// TIA Portal V16 export
// export: Created 2023-03-29T11:03:28.4713144Z, ExportSetting WithDefaults, DisplayName Totally Integrated Automation Portal, DisplayVersion V16 Update 6, DisplayName TIA Portal Version Control Interface, DisplayVersion V16 Update 2, DisplayName TIA Portal Openness, DisplayVersion V16 Update 6, DisplayName STEP 7 Professional, DisplayVersion V16 Update 6, DisplayName STEP 7 Safety, DisplayVersion V16, DisplayName WinCC Advanced, DisplayVersion V16 Update 6
FUNCTION "Synchroniczna_wymiana_danych_PLC1-PLC2" : Void   // FC34, LAD
TITLE = Przekazywanie zmian parametrów
{ S7_Optimized_Access := 'TRUE' }
AUTHOR : rtecmer
VERSION : 0.1
// Funkcja grupuje bloki funkcji służąc wymianie danych HMI - PLC1, HMI-PLC2 i SCADA. Wprowadzanie wartości z poziomu HMI Zbiorniki lub HMI Pompownia czy SCADA jest nadpisywane w docelowym sterowniku. Zmian włónych parametrów układu sterowania pompownią, zbiornikami można dokonywać w dowolnego miejsca.
// stored: AutoNumber true, IsIECCheckEnabled false, SetENOAutomatically false, UDAEnableTagReadback false
   VAR_TEMP   // added for the SCL form of the ladder/FBD networks
      _w1 : Bool;
   END_VAR
BEGIN

REGION Network 2: Detekcja zmiany wartości nastaw - Pozim napełniania
   // Funkcja po przeprowadzeniu sprawdzenia czy nastąpiły zmiany w danych przekazuje nowe wartości
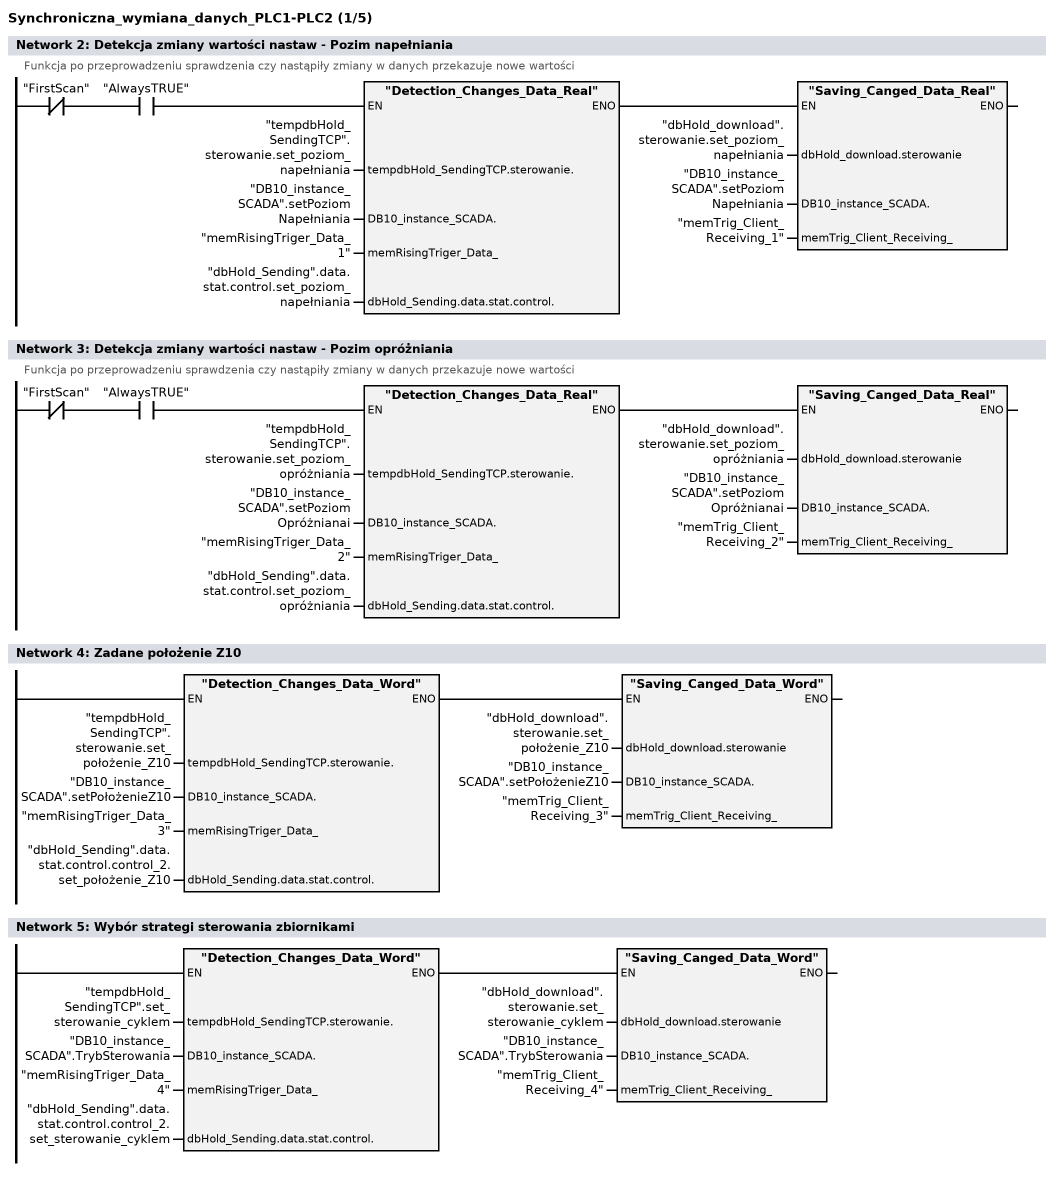
   RUNG wire#powerrail
      I_Contact( "FirstScan" )
      Contact( "AlwaysTRUE" )
      "Detection_Changes_Data_Real"("tempdbHold_SendingTCP.sterowanie." := "tempdbHold_SendingTCP".sterowanie.set_poziom_napełniania, "DB10_instance_SCADA." := "DB10_instance_SCADA".setPoziomNapełniania, memRisingTriger_Data_ := "memRisingTriger_Data_1", "dbHold_Sending.data.stat.control." := "dbHold_Sending".data.stat.control.set_poziom_napełniania)
      "Saving_Canged_Data_Real"("dbHold_download.sterowanie" := "dbHold_download".sterowanie.set_poziom_napełniania, "DB10_instance_SCADA." := "DB10_instance_SCADA".setPoziomNapełniania, memTrig_Client_Receiving_ := "memTrig_Client_Receiving_1")
   END_RUNG
   // the same network as SCL:
   "Detection_Changes_Data_Real"(EN := NOT "FirstScan" AND "AlwaysTRUE",
                           "tempdbHold_SendingTCP.sterowanie." := "tempdbHold_SendingTCP".sterowanie.set_poziom_napełniania,
                           "DB10_instance_SCADA." := "DB10_instance_SCADA".setPoziomNapełniania,
                           memRisingTriger_Data_ := "memRisingTriger_Data_1",
                           "dbHold_Sending.data.stat.control." := "dbHold_Sending".data.stat.control.set_poziom_napełniania,
                           ENO => #_w1);
   IF #_w1 THEN
       "Saving_Canged_Data_Real"("dbHold_download.sterowanie" := "dbHold_download".sterowanie.set_poziom_napełniania,
                               "DB10_instance_SCADA." := "DB10_instance_SCADA".setPoziomNapełniania,
                               memTrig_Client_Receiving_ := "memTrig_Client_Receiving_1");
   END_IF;
END_REGION

REGION Network 3: Detekcja zmiany wartości nastaw - Pozim opróżniania
   // Funkcja po przeprowadzeniu sprawdzenia czy nastąpiły zmiany w danych przekazuje nowe wartości
   RUNG wire#powerrail
      I_Contact( "FirstScan" )
      Contact( "AlwaysTRUE" )
      "Detection_Changes_Data_Real"("tempdbHold_SendingTCP.sterowanie." := "tempdbHold_SendingTCP".sterowanie.set_poziom_opróżniania, "DB10_instance_SCADA." := "DB10_instance_SCADA".setPoziomOpróżnianai, memRisingTriger_Data_ := "memRisingTriger_Data_2", "dbHold_Sending.data.stat.control." := "dbHold_Sending".data.stat.control.set_poziom_opróżniania)
      "Saving_Canged_Data_Real"("dbHold_download.sterowanie" := "dbHold_download".sterowanie.set_poziom_opróżniania, "DB10_instance_SCADA." := "DB10_instance_SCADA".setPoziomOpróżnianai, memTrig_Client_Receiving_ := "memTrig_Client_Receiving_2")
   END_RUNG
   // the same network as SCL:
   "Detection_Changes_Data_Real"(EN := NOT "FirstScan" AND "AlwaysTRUE",
                           "tempdbHold_SendingTCP.sterowanie." := "tempdbHold_SendingTCP".sterowanie.set_poziom_opróżniania,
                           "DB10_instance_SCADA." := "DB10_instance_SCADA".setPoziomOpróżnianai,
                           memRisingTriger_Data_ := "memRisingTriger_Data_2",
                           "dbHold_Sending.data.stat.control." := "dbHold_Sending".data.stat.control.set_poziom_opróżniania,
                           ENO => #_w1);
   IF #_w1 THEN
       "Saving_Canged_Data_Real"("dbHold_download.sterowanie" := "dbHold_download".sterowanie.set_poziom_opróżniania,
                               "DB10_instance_SCADA." := "DB10_instance_SCADA".setPoziomOpróżnianai,
                               memTrig_Client_Receiving_ := "memTrig_Client_Receiving_2");
   END_IF;
END_REGION

REGION Network 4: Zadane położenie Z10
   RUNG wire#powerrail
      "Detection_Changes_Data_Word"("tempdbHold_SendingTCP.sterowanie." := "tempdbHold_SendingTCP".sterowanie.set_położenie_Z10, "DB10_instance_SCADA." := "DB10_instance_SCADA".setPołożenieZ10, memRisingTriger_Data_ := "memRisingTriger_Data_3", "dbHold_Sending.data.stat.control." := "dbHold_Sending".data.stat.control.control_2.set_położenie_Z10)
      "Saving_Canged_Data_Word"("dbHold_download.sterowanie" := "dbHold_download".sterowanie.set_położenie_Z10, "DB10_instance_SCADA." := "DB10_instance_SCADA".setPołożenieZ10, memTrig_Client_Receiving_ := "memTrig_Client_Receiving_3")
   END_RUNG
   // the same network as SCL:
   "Detection_Changes_Data_Word"("tempdbHold_SendingTCP.sterowanie." := "tempdbHold_SendingTCP".sterowanie.set_położenie_Z10,
                           "DB10_instance_SCADA." := "DB10_instance_SCADA".setPołożenieZ10,
                           memRisingTriger_Data_ := "memRisingTriger_Data_3",
                           "dbHold_Sending.data.stat.control." := "dbHold_Sending".data.stat.control.control_2.set_położenie_Z10,
                           ENO => #_w1);
   IF #_w1 THEN
       "Saving_Canged_Data_Word"("dbHold_download.sterowanie" := "dbHold_download".sterowanie.set_położenie_Z10,
                               "DB10_instance_SCADA." := "DB10_instance_SCADA".setPołożenieZ10,
                               memTrig_Client_Receiving_ := "memTrig_Client_Receiving_3");
   END_IF;
END_REGION

REGION Network 5: Wybór strategi sterowania zbiornikami
   RUNG wire#powerrail
      "Detection_Changes_Data_Word"("tempdbHold_SendingTCP.sterowanie." := "tempdbHold_SendingTCP".set_sterowanie_cyklem, "DB10_instance_SCADA." := "DB10_instance_SCADA".TrybSterowania, memRisingTriger_Data_ := "memRisingTriger_Data_4", "dbHold_Sending.data.stat.control." := "dbHold_Sending".data.stat.control.control_2.set_sterowanie_cyklem)
      "Saving_Canged_Data_Word"("dbHold_download.sterowanie" := "dbHold_download".sterowanie.set_sterowanie_cyklem, "DB10_instance_SCADA." := "DB10_instance_SCADA".TrybSterowania, memTrig_Client_Receiving_ := "memTrig_Client_Receiving_4")
   END_RUNG
   // the same network as SCL:
   "Detection_Changes_Data_Word"("tempdbHold_SendingTCP.sterowanie." := "tempdbHold_SendingTCP".set_sterowanie_cyklem,
                           "DB10_instance_SCADA." := "DB10_instance_SCADA".TrybSterowania,
                           memRisingTriger_Data_ := "memRisingTriger_Data_4",
                           "dbHold_Sending.data.stat.control." := "dbHold_Sending".data.stat.control.control_2.set_sterowanie_cyklem,
                           ENO => #_w1);
   IF #_w1 THEN
       "Saving_Canged_Data_Word"("dbHold_download.sterowanie" := "dbHold_download".sterowanie.set_sterowanie_cyklem,
                               "DB10_instance_SCADA." := "DB10_instance_SCADA".TrybSterowania,
                               memTrig_Client_Receiving_ := "memTrig_Client_Receiving_4");
   END_IF;
END_REGION

REGION Network 6: Godzina start napełnianie
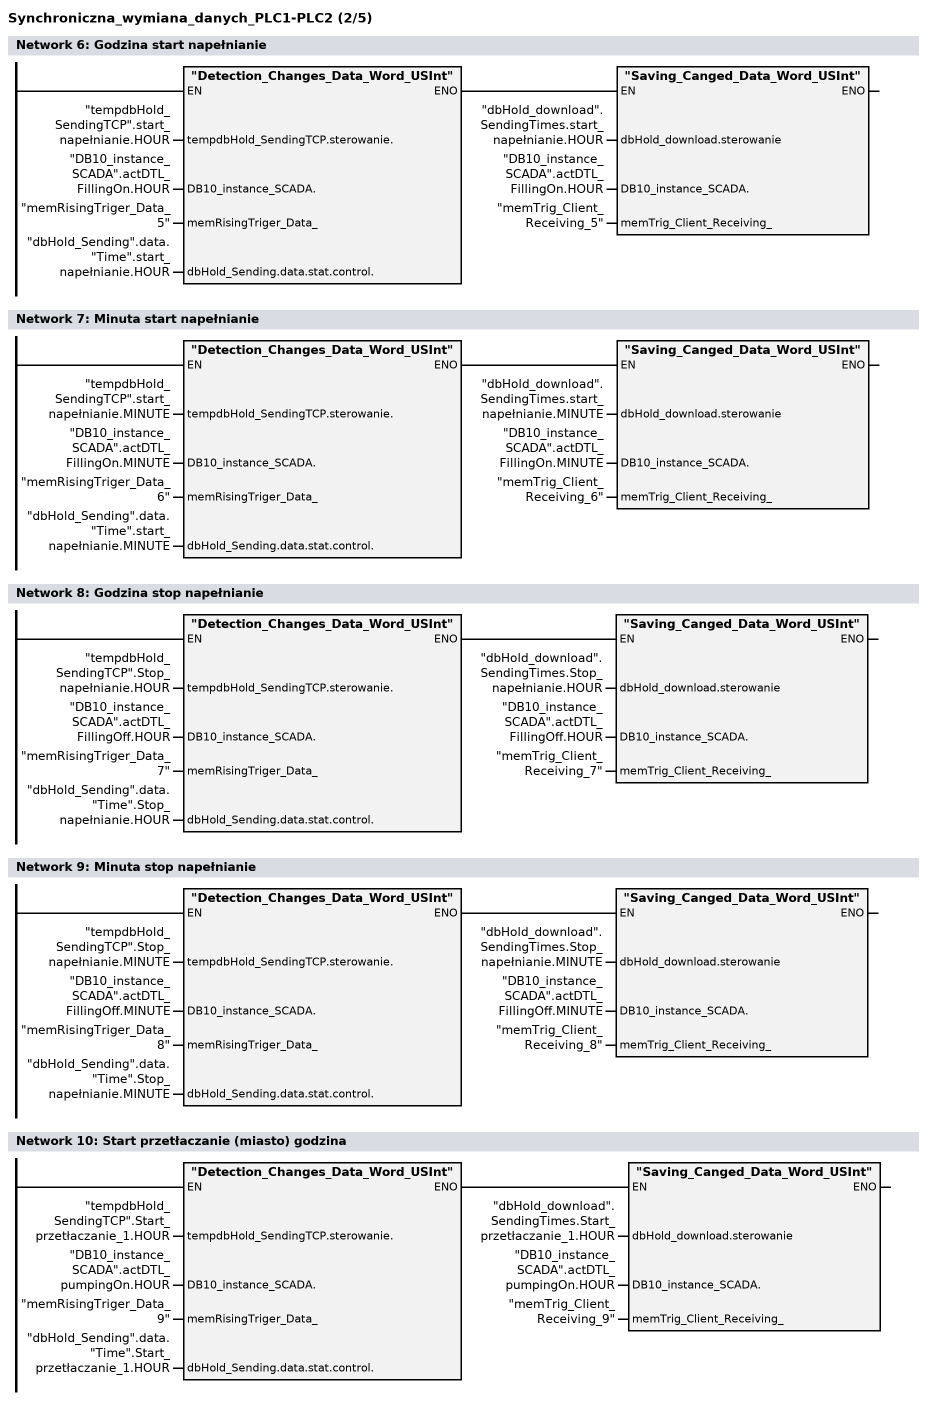
   RUNG wire#powerrail
      "Detection_Changes_Data_Word_USInt"("tempdbHold_SendingTCP.sterowanie." := "tempdbHold_SendingTCP".start_napełnianie.HOUR, "DB10_instance_SCADA." := "DB10_instance_SCADA".actDTL_FillingOn.HOUR, memRisingTriger_Data_ := "memRisingTriger_Data_5", "dbHold_Sending.data.stat.control." := "dbHold_Sending".data."Time".start_napełnianie.HOUR)
      "Saving_Canged_Data_Word_USInt"("dbHold_download.sterowanie" := "dbHold_download".SendingTimes.start_napełnianie.HOUR, "DB10_instance_SCADA." := "DB10_instance_SCADA".actDTL_FillingOn.HOUR, memTrig_Client_Receiving_ := "memTrig_Client_Receiving_5")
   END_RUNG
   // the same network as SCL:
   "Detection_Changes_Data_Word_USInt"("tempdbHold_SendingTCP.sterowanie." := "tempdbHold_SendingTCP".start_napełnianie.HOUR,
                           "DB10_instance_SCADA." := "DB10_instance_SCADA".actDTL_FillingOn.HOUR,
                           memRisingTriger_Data_ := "memRisingTriger_Data_5",
                           "dbHold_Sending.data.stat.control." := "dbHold_Sending".data."Time".start_napełnianie.HOUR,
                           ENO => #_w1);
   IF #_w1 THEN
       "Saving_Canged_Data_Word_USInt"("dbHold_download.sterowanie" := "dbHold_download".SendingTimes.start_napełnianie.HOUR,
                               "DB10_instance_SCADA." := "DB10_instance_SCADA".actDTL_FillingOn.HOUR,
                               memTrig_Client_Receiving_ := "memTrig_Client_Receiving_5");
   END_IF;
END_REGION

REGION Network 7: Minuta start napełnianie
   RUNG wire#powerrail
      "Detection_Changes_Data_Word_USInt"("tempdbHold_SendingTCP.sterowanie." := "tempdbHold_SendingTCP".start_napełnianie.MINUTE, "DB10_instance_SCADA." := "DB10_instance_SCADA".actDTL_FillingOn.MINUTE, memRisingTriger_Data_ := "memRisingTriger_Data_6", "dbHold_Sending.data.stat.control." := "dbHold_Sending".data."Time".start_napełnianie.MINUTE)
      "Saving_Canged_Data_Word_USInt"("dbHold_download.sterowanie" := "dbHold_download".SendingTimes.start_napełnianie.MINUTE, "DB10_instance_SCADA." := "DB10_instance_SCADA".actDTL_FillingOn.MINUTE, memTrig_Client_Receiving_ := "memTrig_Client_Receiving_6")
   END_RUNG
   // the same network as SCL:
   "Detection_Changes_Data_Word_USInt"("tempdbHold_SendingTCP.sterowanie." := "tempdbHold_SendingTCP".start_napełnianie.MINUTE,
                           "DB10_instance_SCADA." := "DB10_instance_SCADA".actDTL_FillingOn.MINUTE,
                           memRisingTriger_Data_ := "memRisingTriger_Data_6",
                           "dbHold_Sending.data.stat.control." := "dbHold_Sending".data."Time".start_napełnianie.MINUTE,
                           ENO => #_w1);
   IF #_w1 THEN
       "Saving_Canged_Data_Word_USInt"("dbHold_download.sterowanie" := "dbHold_download".SendingTimes.start_napełnianie.MINUTE,
                               "DB10_instance_SCADA." := "DB10_instance_SCADA".actDTL_FillingOn.MINUTE,
                               memTrig_Client_Receiving_ := "memTrig_Client_Receiving_6");
   END_IF;
END_REGION

REGION Network 8: Godzina stop napełnianie
   RUNG wire#powerrail
      "Detection_Changes_Data_Word_USInt"("tempdbHold_SendingTCP.sterowanie." := "tempdbHold_SendingTCP".Stop_napełnianie.HOUR, "DB10_instance_SCADA." := "DB10_instance_SCADA".actDTL_FillingOff.HOUR, memRisingTriger_Data_ := "memRisingTriger_Data_7", "dbHold_Sending.data.stat.control." := "dbHold_Sending".data."Time".Stop_napełnianie.HOUR)
      "Saving_Canged_Data_Word_USInt"("dbHold_download.sterowanie" := "dbHold_download".SendingTimes.Stop_napełnianie.HOUR, "DB10_instance_SCADA." := "DB10_instance_SCADA".actDTL_FillingOff.HOUR, memTrig_Client_Receiving_ := "memTrig_Client_Receiving_7")
   END_RUNG
   // the same network as SCL:
   "Detection_Changes_Data_Word_USInt"("tempdbHold_SendingTCP.sterowanie." := "tempdbHold_SendingTCP".Stop_napełnianie.HOUR,
                           "DB10_instance_SCADA." := "DB10_instance_SCADA".actDTL_FillingOff.HOUR,
                           memRisingTriger_Data_ := "memRisingTriger_Data_7",
                           "dbHold_Sending.data.stat.control." := "dbHold_Sending".data."Time".Stop_napełnianie.HOUR,
                           ENO => #_w1);
   IF #_w1 THEN
       "Saving_Canged_Data_Word_USInt"("dbHold_download.sterowanie" := "dbHold_download".SendingTimes.Stop_napełnianie.HOUR,
                               "DB10_instance_SCADA." := "DB10_instance_SCADA".actDTL_FillingOff.HOUR,
                               memTrig_Client_Receiving_ := "memTrig_Client_Receiving_7");
   END_IF;
END_REGION

REGION Network 9: Minuta stop napełnianie
   RUNG wire#powerrail
      "Detection_Changes_Data_Word_USInt"("tempdbHold_SendingTCP.sterowanie." := "tempdbHold_SendingTCP".Stop_napełnianie.MINUTE, "DB10_instance_SCADA." := "DB10_instance_SCADA".actDTL_FillingOff.MINUTE, memRisingTriger_Data_ := "memRisingTriger_Data_8", "dbHold_Sending.data.stat.control." := "dbHold_Sending".data."Time".Stop_napełnianie.MINUTE)
      "Saving_Canged_Data_Word_USInt"("dbHold_download.sterowanie" := "dbHold_download".SendingTimes.Stop_napełnianie.MINUTE, "DB10_instance_SCADA." := "DB10_instance_SCADA".actDTL_FillingOff.MINUTE, memTrig_Client_Receiving_ := "memTrig_Client_Receiving_8")
   END_RUNG
   // the same network as SCL:
   "Detection_Changes_Data_Word_USInt"("tempdbHold_SendingTCP.sterowanie." := "tempdbHold_SendingTCP".Stop_napełnianie.MINUTE,
                           "DB10_instance_SCADA." := "DB10_instance_SCADA".actDTL_FillingOff.MINUTE,
                           memRisingTriger_Data_ := "memRisingTriger_Data_8",
                           "dbHold_Sending.data.stat.control." := "dbHold_Sending".data."Time".Stop_napełnianie.MINUTE,
                           ENO => #_w1);
   IF #_w1 THEN
       "Saving_Canged_Data_Word_USInt"("dbHold_download.sterowanie" := "dbHold_download".SendingTimes.Stop_napełnianie.MINUTE,
                               "DB10_instance_SCADA." := "DB10_instance_SCADA".actDTL_FillingOff.MINUTE,
                               memTrig_Client_Receiving_ := "memTrig_Client_Receiving_8");
   END_IF;
END_REGION

REGION Network 10: Start przetłaczanie (miasto) godzina
   RUNG wire#powerrail
      "Detection_Changes_Data_Word_USInt"("tempdbHold_SendingTCP.sterowanie." := "tempdbHold_SendingTCP".Start_przetłaczanie_1.HOUR, "DB10_instance_SCADA." := "DB10_instance_SCADA".actDTL_pumpingOn.HOUR, memRisingTriger_Data_ := "memRisingTriger_Data_9", "dbHold_Sending.data.stat.control." := "dbHold_Sending".data."Time".Start_przetłaczanie_1.HOUR)
      "Saving_Canged_Data_Word_USInt"("dbHold_download.sterowanie" := "dbHold_download".SendingTimes.Start_przetłaczanie_1.HOUR, "DB10_instance_SCADA." := "DB10_instance_SCADA".actDTL_pumpingOn.HOUR, memTrig_Client_Receiving_ := "memTrig_Client_Receiving_9")
   END_RUNG
   // the same network as SCL:
   "Detection_Changes_Data_Word_USInt"("tempdbHold_SendingTCP.sterowanie." := "tempdbHold_SendingTCP".Start_przetłaczanie_1.HOUR,
                           "DB10_instance_SCADA." := "DB10_instance_SCADA".actDTL_pumpingOn.HOUR,
                           memRisingTriger_Data_ := "memRisingTriger_Data_9",
                           "dbHold_Sending.data.stat.control." := "dbHold_Sending".data."Time".Start_przetłaczanie_1.HOUR,
                           ENO => #_w1);
   IF #_w1 THEN
       "Saving_Canged_Data_Word_USInt"("dbHold_download.sterowanie" := "dbHold_download".SendingTimes.Start_przetłaczanie_1.HOUR,
                               "DB10_instance_SCADA." := "DB10_instance_SCADA".actDTL_pumpingOn.HOUR,
                               memTrig_Client_Receiving_ := "memTrig_Client_Receiving_9");
   END_IF;
END_REGION

REGION Network 11: Start przetłaczanie (miasto) mnutya
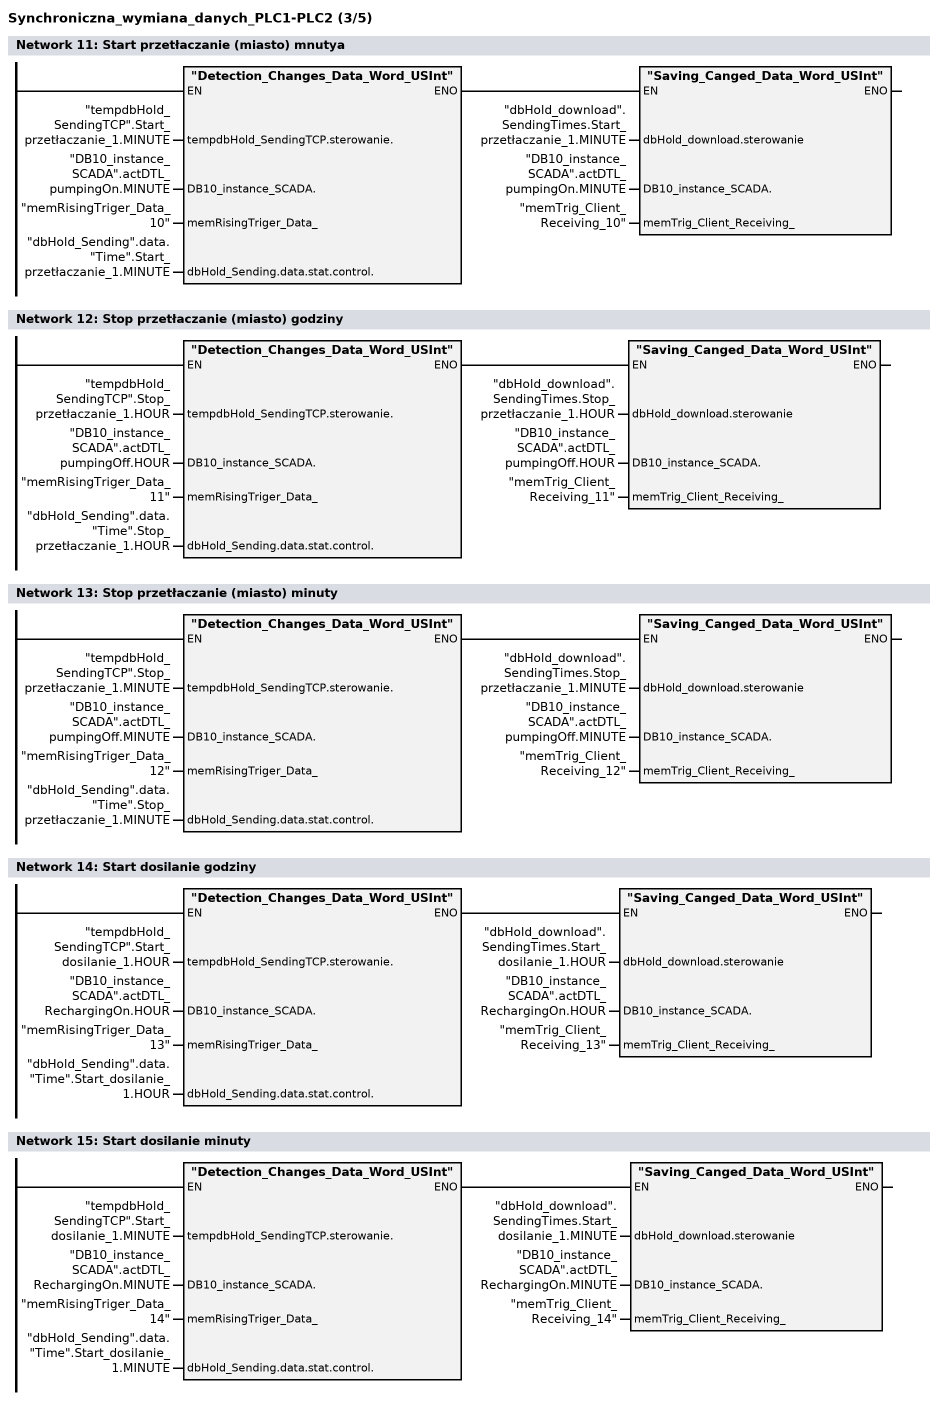
   RUNG wire#powerrail
      "Detection_Changes_Data_Word_USInt"("tempdbHold_SendingTCP.sterowanie." := "tempdbHold_SendingTCP".Start_przetłaczanie_1.MINUTE, "DB10_instance_SCADA." := "DB10_instance_SCADA".actDTL_pumpingOn.MINUTE, memRisingTriger_Data_ := "memRisingTriger_Data_10", "dbHold_Sending.data.stat.control." := "dbHold_Sending".data."Time".Start_przetłaczanie_1.MINUTE)
      "Saving_Canged_Data_Word_USInt"("dbHold_download.sterowanie" := "dbHold_download".SendingTimes.Start_przetłaczanie_1.MINUTE, "DB10_instance_SCADA." := "DB10_instance_SCADA".actDTL_pumpingOn.MINUTE, memTrig_Client_Receiving_ := "memTrig_Client_Receiving_10")
   END_RUNG
   // the same network as SCL:
   "Detection_Changes_Data_Word_USInt"("tempdbHold_SendingTCP.sterowanie." := "tempdbHold_SendingTCP".Start_przetłaczanie_1.MINUTE,
                           "DB10_instance_SCADA." := "DB10_instance_SCADA".actDTL_pumpingOn.MINUTE,
                           memRisingTriger_Data_ := "memRisingTriger_Data_10",
                           "dbHold_Sending.data.stat.control." := "dbHold_Sending".data."Time".Start_przetłaczanie_1.MINUTE,
                           ENO => #_w1);
   IF #_w1 THEN
       "Saving_Canged_Data_Word_USInt"("dbHold_download.sterowanie" := "dbHold_download".SendingTimes.Start_przetłaczanie_1.MINUTE,
                               "DB10_instance_SCADA." := "DB10_instance_SCADA".actDTL_pumpingOn.MINUTE,
                               memTrig_Client_Receiving_ := "memTrig_Client_Receiving_10");
   END_IF;
END_REGION

REGION Network 12: Stop przetłaczanie (miasto) godziny
   RUNG wire#powerrail
      "Detection_Changes_Data_Word_USInt"("tempdbHold_SendingTCP.sterowanie." := "tempdbHold_SendingTCP".Stop_przetłaczanie_1.HOUR, "DB10_instance_SCADA." := "DB10_instance_SCADA".actDTL_pumpingOff.HOUR, memRisingTriger_Data_ := "memRisingTriger_Data_11", "dbHold_Sending.data.stat.control." := "dbHold_Sending".data."Time".Stop_przetłaczanie_1.HOUR)
      "Saving_Canged_Data_Word_USInt"("dbHold_download.sterowanie" := "dbHold_download".SendingTimes.Stop_przetłaczanie_1.HOUR, "DB10_instance_SCADA." := "DB10_instance_SCADA".actDTL_pumpingOff.HOUR, memTrig_Client_Receiving_ := "memTrig_Client_Receiving_11")
   END_RUNG
   // the same network as SCL:
   "Detection_Changes_Data_Word_USInt"("tempdbHold_SendingTCP.sterowanie." := "tempdbHold_SendingTCP".Stop_przetłaczanie_1.HOUR,
                           "DB10_instance_SCADA." := "DB10_instance_SCADA".actDTL_pumpingOff.HOUR,
                           memRisingTriger_Data_ := "memRisingTriger_Data_11",
                           "dbHold_Sending.data.stat.control." := "dbHold_Sending".data."Time".Stop_przetłaczanie_1.HOUR,
                           ENO => #_w1);
   IF #_w1 THEN
       "Saving_Canged_Data_Word_USInt"("dbHold_download.sterowanie" := "dbHold_download".SendingTimes.Stop_przetłaczanie_1.HOUR,
                               "DB10_instance_SCADA." := "DB10_instance_SCADA".actDTL_pumpingOff.HOUR,
                               memTrig_Client_Receiving_ := "memTrig_Client_Receiving_11");
   END_IF;
END_REGION

REGION Network 13: Stop przetłaczanie (miasto) minuty
   RUNG wire#powerrail
      "Detection_Changes_Data_Word_USInt"("tempdbHold_SendingTCP.sterowanie." := "tempdbHold_SendingTCP".Stop_przetłaczanie_1.MINUTE, "DB10_instance_SCADA." := "DB10_instance_SCADA".actDTL_pumpingOff.MINUTE, memRisingTriger_Data_ := "memRisingTriger_Data_12", "dbHold_Sending.data.stat.control." := "dbHold_Sending".data."Time".Stop_przetłaczanie_1.MINUTE)
      "Saving_Canged_Data_Word_USInt"("dbHold_download.sterowanie" := "dbHold_download".SendingTimes.Stop_przetłaczanie_1.MINUTE, "DB10_instance_SCADA." := "DB10_instance_SCADA".actDTL_pumpingOff.MINUTE, memTrig_Client_Receiving_ := "memTrig_Client_Receiving_12")
   END_RUNG
   // the same network as SCL:
   "Detection_Changes_Data_Word_USInt"("tempdbHold_SendingTCP.sterowanie." := "tempdbHold_SendingTCP".Stop_przetłaczanie_1.MINUTE,
                           "DB10_instance_SCADA." := "DB10_instance_SCADA".actDTL_pumpingOff.MINUTE,
                           memRisingTriger_Data_ := "memRisingTriger_Data_12",
                           "dbHold_Sending.data.stat.control." := "dbHold_Sending".data."Time".Stop_przetłaczanie_1.MINUTE,
                           ENO => #_w1);
   IF #_w1 THEN
       "Saving_Canged_Data_Word_USInt"("dbHold_download.sterowanie" := "dbHold_download".SendingTimes.Stop_przetłaczanie_1.MINUTE,
                               "DB10_instance_SCADA." := "DB10_instance_SCADA".actDTL_pumpingOff.MINUTE,
                               memTrig_Client_Receiving_ := "memTrig_Client_Receiving_12");
   END_IF;
END_REGION

REGION Network 14: Start dosilanie godziny
   RUNG wire#powerrail
      "Detection_Changes_Data_Word_USInt"("tempdbHold_SendingTCP.sterowanie." := "tempdbHold_SendingTCP".Start_dosilanie_1.HOUR, "DB10_instance_SCADA." := "DB10_instance_SCADA".actDTL_RechargingOn.HOUR, memRisingTriger_Data_ := "memRisingTriger_Data_13", "dbHold_Sending.data.stat.control." := "dbHold_Sending".data."Time".Start_dosilanie_1.HOUR)
      "Saving_Canged_Data_Word_USInt"("dbHold_download.sterowanie" := "dbHold_download".SendingTimes.Start_dosilanie_1.HOUR, "DB10_instance_SCADA." := "DB10_instance_SCADA".actDTL_RechargingOn.HOUR, memTrig_Client_Receiving_ := "memTrig_Client_Receiving_13")
   END_RUNG
   // the same network as SCL:
   "Detection_Changes_Data_Word_USInt"("tempdbHold_SendingTCP.sterowanie." := "tempdbHold_SendingTCP".Start_dosilanie_1.HOUR,
                           "DB10_instance_SCADA." := "DB10_instance_SCADA".actDTL_RechargingOn.HOUR,
                           memRisingTriger_Data_ := "memRisingTriger_Data_13",
                           "dbHold_Sending.data.stat.control." := "dbHold_Sending".data."Time".Start_dosilanie_1.HOUR,
                           ENO => #_w1);
   IF #_w1 THEN
       "Saving_Canged_Data_Word_USInt"("dbHold_download.sterowanie" := "dbHold_download".SendingTimes.Start_dosilanie_1.HOUR,
                               "DB10_instance_SCADA." := "DB10_instance_SCADA".actDTL_RechargingOn.HOUR,
                               memTrig_Client_Receiving_ := "memTrig_Client_Receiving_13");
   END_IF;
END_REGION

REGION Network 15: Start dosilanie minuty
   RUNG wire#powerrail
      "Detection_Changes_Data_Word_USInt"("tempdbHold_SendingTCP.sterowanie." := "tempdbHold_SendingTCP".Start_dosilanie_1.MINUTE, "DB10_instance_SCADA." := "DB10_instance_SCADA".actDTL_RechargingOn.MINUTE, memRisingTriger_Data_ := "memRisingTriger_Data_14", "dbHold_Sending.data.stat.control." := "dbHold_Sending".data."Time".Start_dosilanie_1.MINUTE)
      "Saving_Canged_Data_Word_USInt"("dbHold_download.sterowanie" := "dbHold_download".SendingTimes.Start_dosilanie_1.MINUTE, "DB10_instance_SCADA." := "DB10_instance_SCADA".actDTL_RechargingOn.MINUTE, memTrig_Client_Receiving_ := "memTrig_Client_Receiving_14")
   END_RUNG
   // the same network as SCL:
   "Detection_Changes_Data_Word_USInt"("tempdbHold_SendingTCP.sterowanie." := "tempdbHold_SendingTCP".Start_dosilanie_1.MINUTE,
                           "DB10_instance_SCADA." := "DB10_instance_SCADA".actDTL_RechargingOn.MINUTE,
                           memRisingTriger_Data_ := "memRisingTriger_Data_14",
                           "dbHold_Sending.data.stat.control." := "dbHold_Sending".data."Time".Start_dosilanie_1.MINUTE,
                           ENO => #_w1);
   IF #_w1 THEN
       "Saving_Canged_Data_Word_USInt"("dbHold_download.sterowanie" := "dbHold_download".SendingTimes.Start_dosilanie_1.MINUTE,
                               "DB10_instance_SCADA." := "DB10_instance_SCADA".actDTL_RechargingOn.MINUTE,
                               memTrig_Client_Receiving_ := "memTrig_Client_Receiving_14");
   END_IF;
END_REGION

REGION Network 16: Stop dosilanie godziny
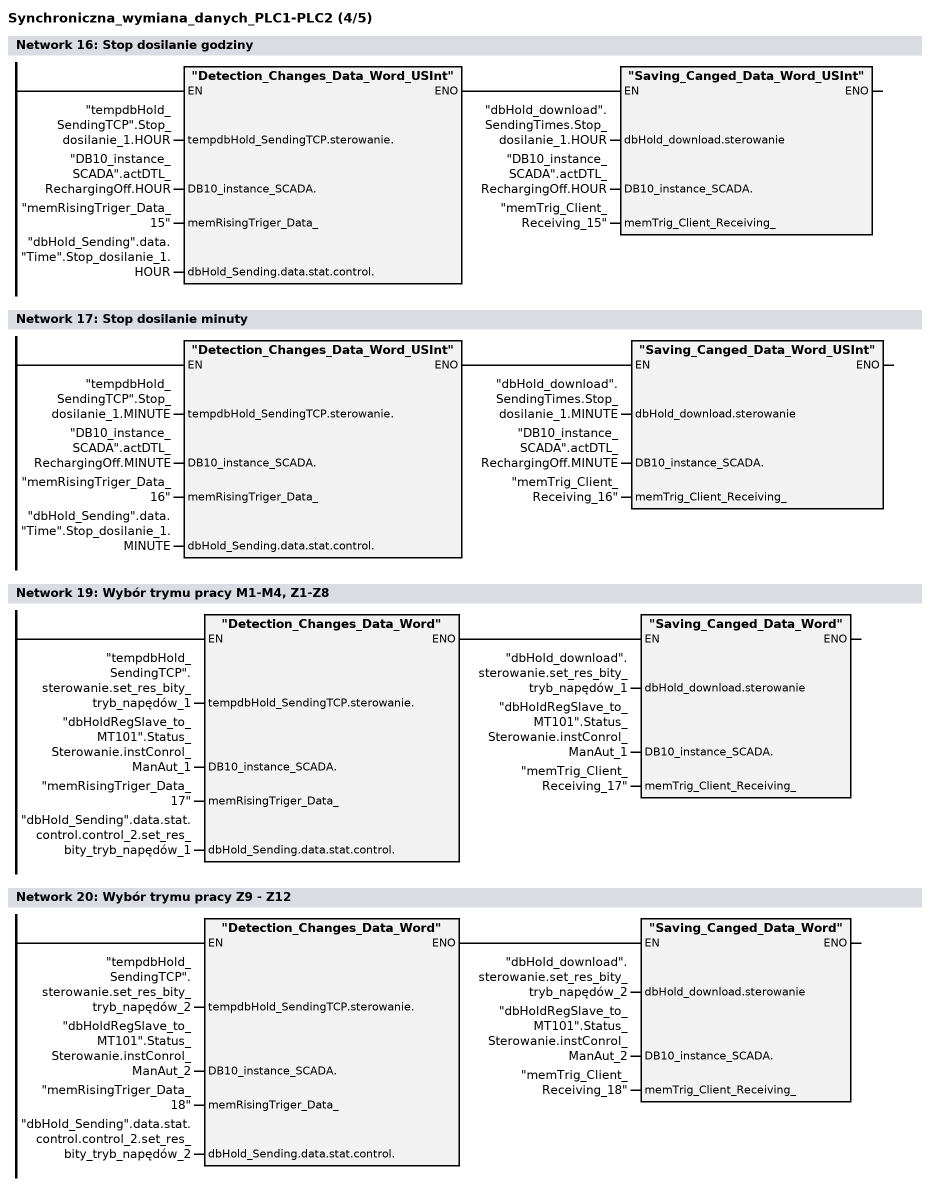
   RUNG wire#powerrail
      "Detection_Changes_Data_Word_USInt"("tempdbHold_SendingTCP.sterowanie." := "tempdbHold_SendingTCP".Stop_dosilanie_1.HOUR, "DB10_instance_SCADA." := "DB10_instance_SCADA".actDTL_RechargingOff.HOUR, memRisingTriger_Data_ := "memRisingTriger_Data_15", "dbHold_Sending.data.stat.control." := "dbHold_Sending".data."Time".Stop_dosilanie_1.HOUR)
      "Saving_Canged_Data_Word_USInt"("dbHold_download.sterowanie" := "dbHold_download".SendingTimes.Stop_dosilanie_1.HOUR, "DB10_instance_SCADA." := "DB10_instance_SCADA".actDTL_RechargingOff.HOUR, memTrig_Client_Receiving_ := "memTrig_Client_Receiving_15")
   END_RUNG
   // the same network as SCL:
   "Detection_Changes_Data_Word_USInt"("tempdbHold_SendingTCP.sterowanie." := "tempdbHold_SendingTCP".Stop_dosilanie_1.HOUR,
                           "DB10_instance_SCADA." := "DB10_instance_SCADA".actDTL_RechargingOff.HOUR,
                           memRisingTriger_Data_ := "memRisingTriger_Data_15",
                           "dbHold_Sending.data.stat.control." := "dbHold_Sending".data."Time".Stop_dosilanie_1.HOUR,
                           ENO => #_w1);
   IF #_w1 THEN
       "Saving_Canged_Data_Word_USInt"("dbHold_download.sterowanie" := "dbHold_download".SendingTimes.Stop_dosilanie_1.HOUR,
                               "DB10_instance_SCADA." := "DB10_instance_SCADA".actDTL_RechargingOff.HOUR,
                               memTrig_Client_Receiving_ := "memTrig_Client_Receiving_15");
   END_IF;
END_REGION

REGION Network 17: Stop dosilanie minuty
   RUNG wire#powerrail
      "Detection_Changes_Data_Word_USInt"("tempdbHold_SendingTCP.sterowanie." := "tempdbHold_SendingTCP".Stop_dosilanie_1.MINUTE, "DB10_instance_SCADA." := "DB10_instance_SCADA".actDTL_RechargingOff.MINUTE, memRisingTriger_Data_ := "memRisingTriger_Data_16", "dbHold_Sending.data.stat.control." := "dbHold_Sending".data."Time".Stop_dosilanie_1.MINUTE)
      "Saving_Canged_Data_Word_USInt"("dbHold_download.sterowanie" := "dbHold_download".SendingTimes.Stop_dosilanie_1.MINUTE, "DB10_instance_SCADA." := "DB10_instance_SCADA".actDTL_RechargingOff.MINUTE, memTrig_Client_Receiving_ := "memTrig_Client_Receiving_16")
   END_RUNG
   // the same network as SCL:
   "Detection_Changes_Data_Word_USInt"("tempdbHold_SendingTCP.sterowanie." := "tempdbHold_SendingTCP".Stop_dosilanie_1.MINUTE,
                           "DB10_instance_SCADA." := "DB10_instance_SCADA".actDTL_RechargingOff.MINUTE,
                           memRisingTriger_Data_ := "memRisingTriger_Data_16",
                           "dbHold_Sending.data.stat.control." := "dbHold_Sending".data."Time".Stop_dosilanie_1.MINUTE,
                           ENO => #_w1);
   IF #_w1 THEN
       "Saving_Canged_Data_Word_USInt"("dbHold_download.sterowanie" := "dbHold_download".SendingTimes.Stop_dosilanie_1.MINUTE,
                               "DB10_instance_SCADA." := "DB10_instance_SCADA".actDTL_RechargingOff.MINUTE,
                               memTrig_Client_Receiving_ := "memTrig_Client_Receiving_16");
   END_IF;
END_REGION

REGION Network 19: Wybór trymu pracy M1-M4, Z1-Z8
   RUNG wire#powerrail
      "Detection_Changes_Data_Word"("tempdbHold_SendingTCP.sterowanie." := "tempdbHold_SendingTCP".sterowanie.set_res_bity_tryb_napędów_1, "DB10_instance_SCADA." := "dbHoldRegSlave_to_MT101".Status_Sterowanie.instConrol_ManAut_1, memRisingTriger_Data_ := "memRisingTriger_Data_17", "dbHold_Sending.data.stat.control." := "dbHold_Sending".data.stat.control.control_2.set_res_bity_tryb_napędów_1)
      "Saving_Canged_Data_Word"("dbHold_download.sterowanie" := "dbHold_download".sterowanie.set_res_bity_tryb_napędów_1, "DB10_instance_SCADA." := "dbHoldRegSlave_to_MT101".Status_Sterowanie.instConrol_ManAut_1, memTrig_Client_Receiving_ := "memTrig_Client_Receiving_17")
   END_RUNG
   // the same network as SCL:
   "Detection_Changes_Data_Word"("tempdbHold_SendingTCP.sterowanie." := "tempdbHold_SendingTCP".sterowanie.set_res_bity_tryb_napędów_1,
                           "DB10_instance_SCADA." := "dbHoldRegSlave_to_MT101".Status_Sterowanie.instConrol_ManAut_1,
                           memRisingTriger_Data_ := "memRisingTriger_Data_17",
                           "dbHold_Sending.data.stat.control." := "dbHold_Sending".data.stat.control.control_2.set_res_bity_tryb_napędów_1,
                           ENO => #_w1);
   IF #_w1 THEN
       "Saving_Canged_Data_Word"("dbHold_download.sterowanie" := "dbHold_download".sterowanie.set_res_bity_tryb_napędów_1,
                               "DB10_instance_SCADA." := "dbHoldRegSlave_to_MT101".Status_Sterowanie.instConrol_ManAut_1,
                               memTrig_Client_Receiving_ := "memTrig_Client_Receiving_17");
   END_IF;
END_REGION

REGION Network 20: Wybór trymu pracy Z9 - Z12
   RUNG wire#powerrail
      "Detection_Changes_Data_Word"("tempdbHold_SendingTCP.sterowanie." := "tempdbHold_SendingTCP".sterowanie.set_res_bity_tryb_napędów_2, "DB10_instance_SCADA." := "dbHoldRegSlave_to_MT101".Status_Sterowanie.instConrol_ManAut_2, memRisingTriger_Data_ := "memRisingTriger_Data_18", "dbHold_Sending.data.stat.control." := "dbHold_Sending".data.stat.control.control_2.set_res_bity_tryb_napędów_2)
      "Saving_Canged_Data_Word"("dbHold_download.sterowanie" := "dbHold_download".sterowanie.set_res_bity_tryb_napędów_2, "DB10_instance_SCADA." := "dbHoldRegSlave_to_MT101".Status_Sterowanie.instConrol_ManAut_2, memTrig_Client_Receiving_ := "memTrig_Client_Receiving_18")
   END_RUNG
   // the same network as SCL:
   "Detection_Changes_Data_Word"("tempdbHold_SendingTCP.sterowanie." := "tempdbHold_SendingTCP".sterowanie.set_res_bity_tryb_napędów_2,
                           "DB10_instance_SCADA." := "dbHoldRegSlave_to_MT101".Status_Sterowanie.instConrol_ManAut_2,
                           memRisingTriger_Data_ := "memRisingTriger_Data_18",
                           "dbHold_Sending.data.stat.control." := "dbHold_Sending".data.stat.control.control_2.set_res_bity_tryb_napędów_2,
                           ENO => #_w1);
   IF #_w1 THEN
       "Saving_Canged_Data_Word"("dbHold_download.sterowanie" := "dbHold_download".sterowanie.set_res_bity_tryb_napędów_2,
                               "DB10_instance_SCADA." := "dbHoldRegSlave_to_MT101".Status_Sterowanie.instConrol_ManAut_2,
                               memTrig_Client_Receiving_ := "memTrig_Client_Receiving_18");
   END_IF;
END_REGION

REGION Network 21: Sterowanie OTWIERANIE/ZAMYKANIE Z1 - Z8
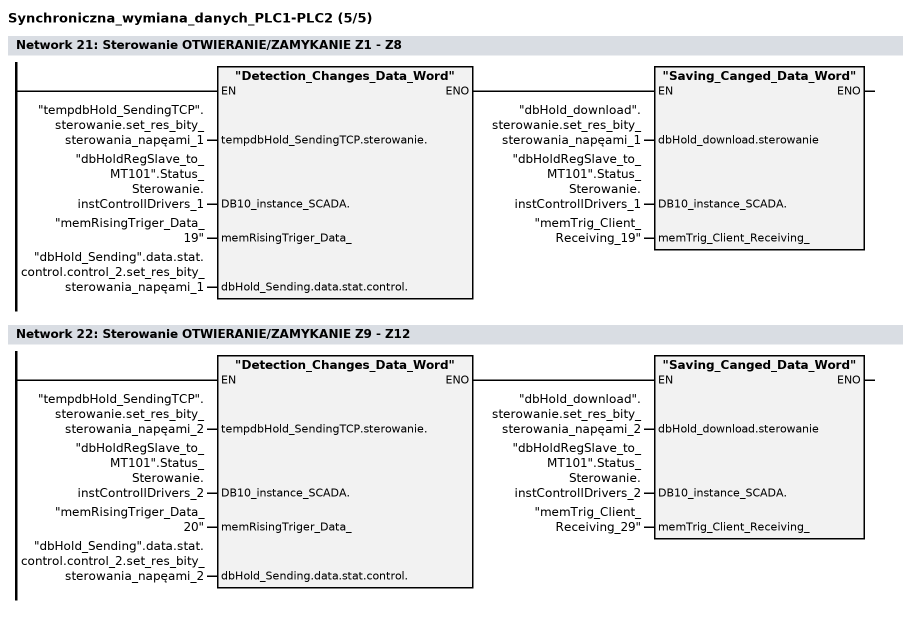
   RUNG wire#powerrail
      "Detection_Changes_Data_Word"("tempdbHold_SendingTCP.sterowanie." := "tempdbHold_SendingTCP".sterowanie.set_res_bity_sterowania_napęami_1, "DB10_instance_SCADA." := "dbHoldRegSlave_to_MT101".Status_Sterowanie.instControllDrivers_1, memRisingTriger_Data_ := "memRisingTriger_Data_19", "dbHold_Sending.data.stat.control." := "dbHold_Sending".data.stat.control.control_2.set_res_bity_sterowania_napęami_1)
      "Saving_Canged_Data_Word"("dbHold_download.sterowanie" := "dbHold_download".sterowanie.set_res_bity_sterowania_napęami_1, "DB10_instance_SCADA." := "dbHoldRegSlave_to_MT101".Status_Sterowanie.instControllDrivers_1, memTrig_Client_Receiving_ := "memTrig_Client_Receiving_19")
   END_RUNG
   // the same network as SCL:
   "Detection_Changes_Data_Word"("tempdbHold_SendingTCP.sterowanie." := "tempdbHold_SendingTCP".sterowanie.set_res_bity_sterowania_napęami_1,
                           "DB10_instance_SCADA." := "dbHoldRegSlave_to_MT101".Status_Sterowanie.instControllDrivers_1,
                           memRisingTriger_Data_ := "memRisingTriger_Data_19",
                           "dbHold_Sending.data.stat.control." := "dbHold_Sending".data.stat.control.control_2.set_res_bity_sterowania_napęami_1,
                           ENO => #_w1);
   IF #_w1 THEN
       "Saving_Canged_Data_Word"("dbHold_download.sterowanie" := "dbHold_download".sterowanie.set_res_bity_sterowania_napęami_1,
                               "DB10_instance_SCADA." := "dbHoldRegSlave_to_MT101".Status_Sterowanie.instControllDrivers_1,
                               memTrig_Client_Receiving_ := "memTrig_Client_Receiving_19");
   END_IF;
END_REGION

REGION Network 22: Sterowanie OTWIERANIE/ZAMYKANIE Z9 - Z12
   RUNG wire#powerrail
      "Detection_Changes_Data_Word"("tempdbHold_SendingTCP.sterowanie." := "tempdbHold_SendingTCP".sterowanie.set_res_bity_sterowania_napęami_2, "DB10_instance_SCADA." := "dbHoldRegSlave_to_MT101".Status_Sterowanie.instControllDrivers_2, memRisingTriger_Data_ := "memRisingTriger_Data_20", "dbHold_Sending.data.stat.control." := "dbHold_Sending".data.stat.control.control_2.set_res_bity_sterowania_napęami_2)
      "Saving_Canged_Data_Word"("dbHold_download.sterowanie" := "dbHold_download".sterowanie.set_res_bity_sterowania_napęami_2, "DB10_instance_SCADA." := "dbHoldRegSlave_to_MT101".Status_Sterowanie.instControllDrivers_2, memTrig_Client_Receiving_ := "memTrig_Client_Receiving_29")
   END_RUNG
   // the same network as SCL:
   "Detection_Changes_Data_Word"("tempdbHold_SendingTCP.sterowanie." := "tempdbHold_SendingTCP".sterowanie.set_res_bity_sterowania_napęami_2,
                           "DB10_instance_SCADA." := "dbHoldRegSlave_to_MT101".Status_Sterowanie.instControllDrivers_2,
                           memRisingTriger_Data_ := "memRisingTriger_Data_20",
                           "dbHold_Sending.data.stat.control." := "dbHold_Sending".data.stat.control.control_2.set_res_bity_sterowania_napęami_2,
                           ENO => #_w1);
   IF #_w1 THEN
       "Saving_Canged_Data_Word"("dbHold_download.sterowanie" := "dbHold_download".sterowanie.set_res_bity_sterowania_napęami_2,
                               "DB10_instance_SCADA." := "dbHoldRegSlave_to_MT101".Status_Sterowanie.instControllDrivers_2,
                               memTrig_Client_Receiving_ := "memTrig_Client_Receiving_29");
   END_IF;
END_REGION
END_FUNCTION
